(* Logix 5000 project; controller DispersionPlc vendor 1 type 14 code 108 rev 34.11; software revision 34.01; part 8 of 22 *)
(* tags used below, declared in another part *)
   Disp_Ons : BOOL[32];
   DispersionProductID_BarcodeScan : STRING;
   DispersionProductID_ScanIndex_Storage : DINT;
   DispersionProductIDEntryStorage : STRING;
   DispersionProductIDMatch : DINT;
   FE_4303_Deaband_Minus : REAL;
   FE_4303_Deaband_Plus : REAL;
   FE_4303_Feed_Error : REAL;
   FE_4303_Temp : REAL;
   Messaging_Timer2 : TIMER;
   MMI_SV4303_01_PB : BOOL;
   MMI_V4303_Acc_weight : REAL;
   MonDispenced_Snapshot : REAL;
   Monomer_FlowTimer : TIMER;
   Monomer_OneShots : BOOL[32];
   Monomer_Target_Wgt_Lb_Min : REAL;
   MonomerTimers : TIMER[12];
   ONS : BOOL[32];
   ons100 : BOOL;
   P4303_Rate : REAL;
   SV_4303_03_Man_Override : BOOL;
   T4301_T4302_Xfer_In_Enable : BOOL;
   W4303_RampTimer : TIMER;
   AFI : BOOL;
   BarcodeBypassAcitve : BOOL;
   BarcodeBypassAcitvePB : BOOL;
   BarcodeForEditString : STRING;
   BarcodeIndex : DINT;
   BarcodeIndex_Hold : DINT;
   BLANK64 : Stp64;
   BlankStrg : STRING;
   Cat_Tank_Destination : DINT;
   Control_Rm_tags : DINT;
   CR : STRING;
   CRADT : ALIAS FOR Local:5:O.Data.7;
   Dispersion_from_Main : DINT;
   Dispersion_from_Main2 : DINT;
   Dispersion_from_Main2_DintToStringConv : STRING;
   Dispersion_from_SIL2 : DINT;
   Dispersion_from_SIL2_Analog : REAL[24];
   Dispersion_to_Main : DINT;
   Dispersion_to_SIL2 : DINT;
   Dispersion_to_SIL2_Analog : REAL[24];
   DispersionAlarms : BOOL[256];
   DispersionProductID : STRING[21];
   DispersionProductID_ScanIndex : DINT;
   DispersionProductIDKeyEntry : STRING;
   DispersionProductIDKeyEntry1 : STRING;
   Drum_Transfer : BOOL;
   Drum_Transfer_Active : BOOL;
   Drum_Transfer_ONS : BOOL;
   Drum_Transfer_ONS_1 : BOOL;
   Enable_High_Alarm : BOOL;
   Enable_Shortstop_Automation : BOOL;
   Estop_Inx : ALIAS FOR Local:3:I.Data.3;
   FE_4303_Corrected : REAL;
   Found : DINT;
   From_Main : MESSAGE;
   From_Sil2 : MESSAGE;
   From_Sil2_Analog : MESSAGE;
   Hold_For_Flow_Switch : BOOL;
   Hold_For_Pump_Enable : BOOL;
   K4_High_Temp : BOOL;
   K4_Low_Temp : BOOL;
   LastScannedCode : STRING;
   LevelAlarmBeaconsRelay : BOOL;
   LS_26_High : BOOL;
   LS_28_H_Alarm : BOOL;
   MAINT_SV4303_03_PB : BOOL;
   MAINT_SV4303_04_PB : BOOL;
   MAINT_XV4303_05_PB : BOOL;
   Messaging_Timer : TIMER;
   MIXER_A_4303_RUN : ALIAS FOR Local:1:O.Data[0].4;
   MMI_A_4303_RUN_PB : BOOL;
   MMI_Mon_Nit_Purge_Time : REAL;
   MMI_Mon_Recirc_Pump_Speed : REAL;
   MMI_P_4303_Run_Pb : BOOL;
   MMI_SV4303_03_PB : BOOL;
   MMI_SV4303_04_PB : BOOL;
   MMI_V4303_Acc_Weight_Reset : BOOL;
   MMI_V4303_TransTime_SP : REAL;
   MMI_V4303_Weight_SP : REAL;
   MMI_W4303_Acc_Weight : REAL;
   MMI_XV4303_03_PB : BOOL;
   MMI_XV4303_04_PB : BOOL;
   MMI_XV4303_05_PB : BOOL;
   Momomer_Ons : DINT;
   Mon_Bogus_Bit : BOOL;
   Mon_Pump_Manual : BOOL;
   Mon_Recirc_Transfer_K400 : Seq64;
   Mon_Recirc_Transfer_T430X : Seq64;
   Mon_Tank_Destination : DINT;
   MON_VALV_ENBL : DINT;
   Monomer_Barcode : STRING;
   Monomer_Barcode_Scan_Index : DINT;
   Monomer_Barcode_Search : BOOL;
   Monomer_Fill_Pump_Running : BOOL;
   Monomer_Fill_Pump_Stopped : BOOL;
   Monomer_Flow_Start_Timer : TIMER;
   Monomer_Flow_Stop_Timer : TIMER;
   Monomer_MaxFeedRate : REAL;
   MONOMER_RESET : BOOL;
   Monomer_Scanner_Reset_Timer : TIMER;
   MonomerTimers_0_HMI : REAL;
   No_Vaild_Monomer_Barcode_Found : BOOL;
   One_Shots : DINT;
   OneShots : DINT;
   Pump_Enable_TMR : TIMER;
   SaveBarcode : BOOL;
   ScreenDisplayBarcode : STRING;
   Shortstop_Activate : BOOL;
   Shortstop_Timer_1 : REAL;
   Shortstop_Timer_2 : REAL;
   SIL2_to_Dispersion : DINT;
   SPARE_O515 : ALIAS FOR Local:5:O.Data.15;
   ST_K400_1 : REAL;
   ST_K400_SAFETY : BOOL;
   SV_4303_01 : ALIAS FOR Local:5:O.Data.8;
   SV_4303_02_ZSC : BOOL;
   SV_4303_02_ZSO : BOOL;
   SV_4303_03 : BOOL;
   SV_4303_03_Enable_PB : BOOL;
   SV_4303_04 : BOOL;
   SV_4303_04_Enable_PB : BOOL;
   T4301_Mixer : VFD;
   T4301_Process_Alarm_Setpoints : Alarm_SPT;
   Task_Permissive : DINT[2];
   TE_4301A : ALIAS FOR Local:8:I.Ch0Data;
   TE_4303_01 : REAL;
   TE_4303_High : REAL;
   To_CtrlRm1 : MESSAGE;
   To_CtrlRm2 : MESSAGE;
   To_CtrlRm3 : MESSAGE;
   To_Main : MESSAGE;
   To_Main2 : MESSAGE;
   To_SIL2 : MESSAGE;
   To_SIL2_Analog : MESSAGE;
   TOGGLE : BOOL;
   TruckLoadLevelAlarmHIHI : BOOL;
   TruckLoadLevelAlarmHIHIRedundant : BOOL;
   TruckLoadLevelAlarmResetPB : BOOL;
   V4304_Pump : VFD;
   Vaild_Monomer_Barcode : BOOL;
   Vaild_Monomer_Barcode_At_Index : DINT;
   Vaild_Monomer_BarcodeS : STRING[20];
   W4303_Pump : VFD;
   XI_K400_1 : BOOL;
   XV_4303_01 : ALIAS FOR Local:5:O.Data.3;
   XV_4303_01_PB : BOOL;
   XV_4303_02_ZSC : BOOL;
   XV_4303_02_ZSO : BOOL;
   XV_4303_03 : BOOL;
   XV_4303_04 : BOOL;
   XV_4303_05 : BOOL;
   XV_K400_03_SEQCLOSE : BOOL;
   XV_K400_03_SEQOPEN : BOOL;
   XV_K400_04_SEQCLOSE : BOOL;
   XV_K400_04_SEQOPEN : BOOL;
   ZSC_4303_03 : BOOL;
   ZSC_4303_04 : BOOL;
   ZSC_4303_05 : BOOL;
   ZSC_4303_1 : ALIAS FOR Local:2:I.Data.7;
   ZSC_K400_03 : BOOL;
   ZSC_K400_04 : BOOL;
   ZSO_4303_04 : BOOL;
   ZSO_4303_05 : BOOL;
   ZSO_K400_03 : BOOL;
   ZSO_K400_04 : BOOL;
(* MainProgram, continued *)

ROUTINE Messaging   (* ladder *)
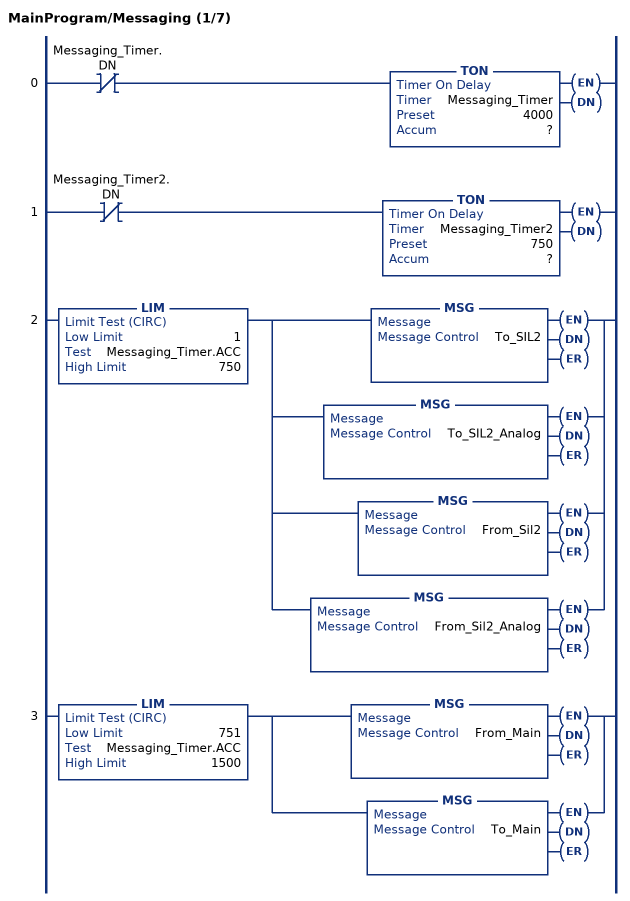
   0: XIO(Messaging_Timer.DN)TON(Messaging_Timer,?,?);
   1: XIO(Messaging_Timer2.DN)TON(Messaging_Timer2,?,?);
   2: LIM(1,Messaging_Timer.ACC,750)[MSG(To_SIL2) ,MSG(To_SIL2_Analog) ,MSG(From_Sil2) ,MSG(From_Sil2_Analog) ];
   3: LIM(751,Messaging_Timer.ACC,1500)[MSG(From_Main) ,MSG(To_Main) ];
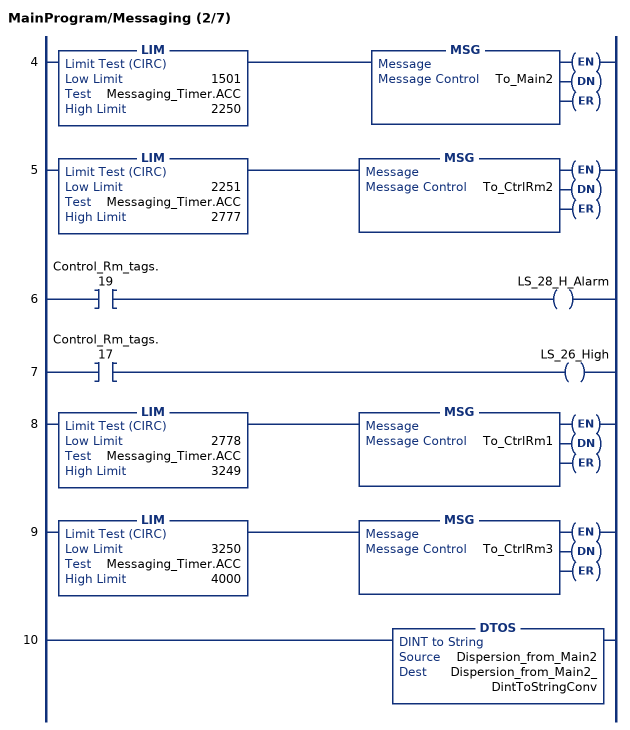
   4: LIM(1501,Messaging_Timer.ACC,2250)MSG(To_Main2);
   5: LIM(2251,Messaging_Timer.ACC,2777)MSG(To_CtrlRm2);
   6: XIC(Control_Rm_tags.19)OTE(LS_28_H_Alarm);
   7: XIC(Control_Rm_tags.17)OTE(LS_26_High);
   8: LIM(2778,Messaging_Timer.ACC,3249)MSG(To_CtrlRm1);
   9: LIM(3250,Messaging_Timer.ACC,4000)MSG(To_CtrlRm3);
   10: DTOS(Dispersion_from_Main2,Dispersion_from_Main2_DintToStringConv);
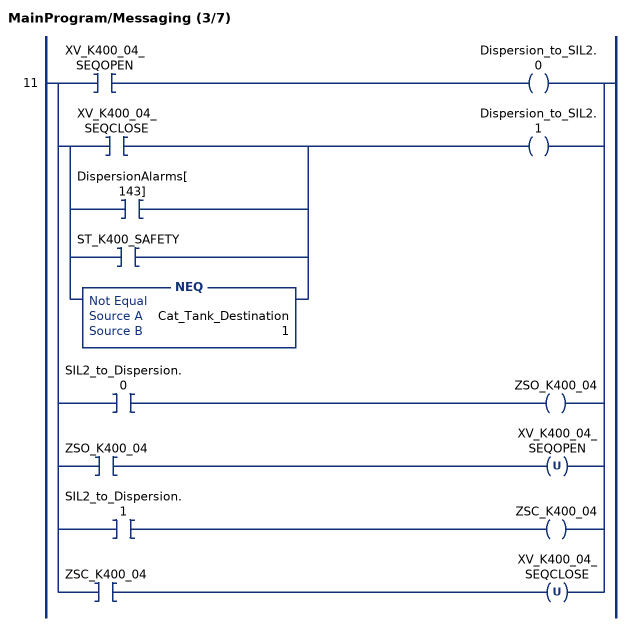
   11: [XIC(XV_K400_04_SEQOPEN) OTE(Dispersion_to_SIL2.0) ,[XIC(XV_K400_04_SEQCLOSE) ,XIC(DispersionAlarms[143]) ,XIC(ST_K400_SAFETY) ,NEQ(Cat_Tank_Destination,1) ] OTE(Dispersion_to_SIL2.1) ,XIC(SIL2_to_Dispersion.0) OTE(ZSO_K400_04) ,XIC(ZSO_K400_04) OTU(XV_K400_04_SEQOPEN) ,XIC(SIL2_to_Dispersion.1) OTE(ZSC_K400_04) ,XIC(ZSC_K400_04) OTU(XV_K400_04_SEQCLOSE) ];
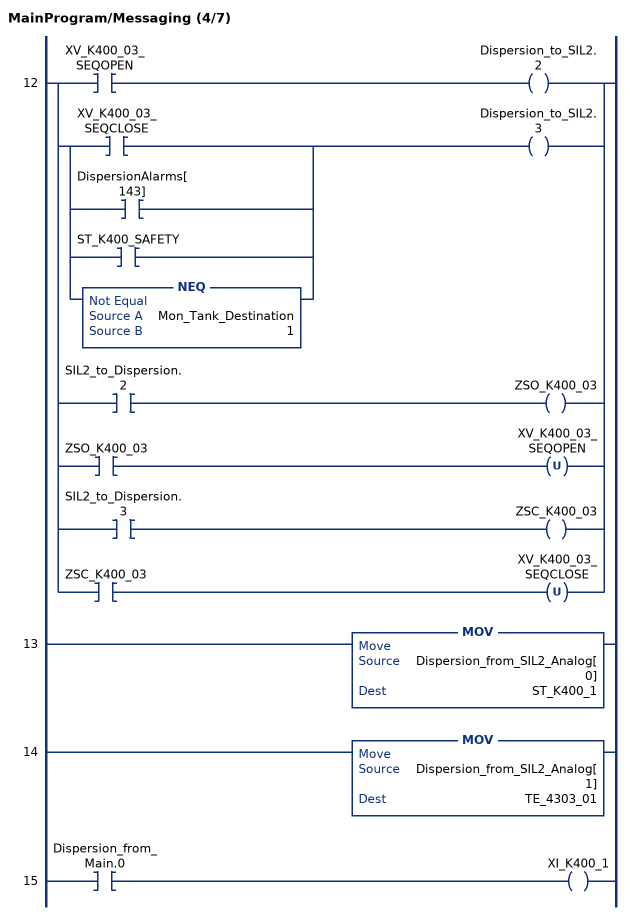
   12: [XIC(XV_K400_03_SEQOPEN) OTE(Dispersion_to_SIL2.2) ,[XIC(XV_K400_03_SEQCLOSE) ,XIC(DispersionAlarms[143]) ,XIC(ST_K400_SAFETY) ,NEQ(Mon_Tank_Destination,1) ] OTE(Dispersion_to_SIL2.3) ,XIC(SIL2_to_Dispersion.2) OTE(ZSO_K400_03) ,XIC(ZSO_K400_03) OTU(XV_K400_03_SEQOPEN) ,XIC(SIL2_to_Dispersion.3) OTE(ZSC_K400_03) ,XIC(ZSC_K400_03) OTU(XV_K400_03_SEQCLOSE) ];
   13: MOV(Dispersion_from_SIL2_Analog[0],ST_K400_1);
   14: MOV(Dispersion_from_SIL2_Analog[1],TE_4303_01);
   15: XIC(Dispersion_from_Main.0)OTE(XI_K400_1);
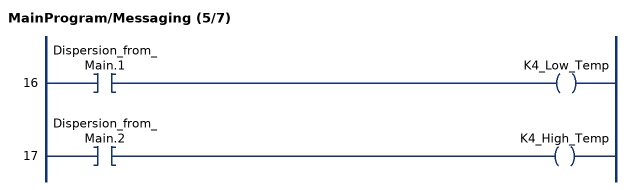
   16: XIC(Dispersion_from_Main.1)OTE(K4_Low_Temp);
   17: XIC(Dispersion_from_Main.2)OTE(K4_High_Temp);
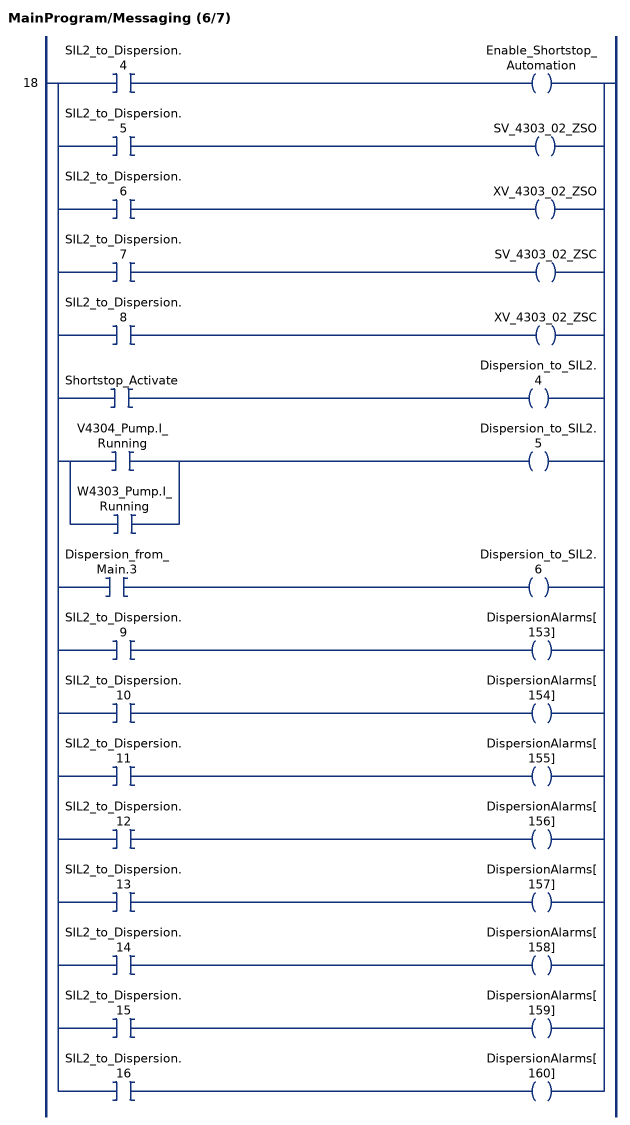
   18: [XIC(SIL2_to_Dispersion.4) OTE(Enable_Shortstop_Automation) ,XIC(SIL2_to_Dispersion.5) OTE(SV_4303_02_ZSO) ,XIC(SIL2_to_Dispersion.6) OTE(XV_4303_02_ZSO) ,XIC(SIL2_to_Dispersion.7) OTE(SV_4303_02_ZSC) ,XIC(SIL2_to_Dispersion.8) OTE(XV_4303_02_ZSC) ,XIC(Shortstop_Activate) OTE(Dispersion_to_SIL2.4) ,[XIC(V4304_Pump.I_Running) ,XIC(W4303_Pump.I_Running) ] OTE(Dispersion_to_SIL2.5) ,XIC(Dispersion_from_Main.3) OTE(Dispersion_to_SIL2.6) ,XIC(SIL2_to_Dispersion.9) OTE(DispersionAlarms[153]) ,XIC(SIL2_to_Dispersion.10) OTE(DispersionAlarms[154]) ,XIC(SIL2_to_Dispersion.11) OTE(DispersionAlarms[155]) ,XIC(SIL2_to_Dispersion.12) OTE(DispersionAlarms[156]) ,XIC(SIL2_to_Dispersion.13) OTE(DispersionAlarms[157]) ,XIC(SIL2_to_Dispersion.14) OTE(DispersionAlarms[158]) ,XIC(SIL2_to_Dispersion.15) OTE(DispersionAlarms[159]) ,XIC(SIL2_to_Dispersion.16) OTE(DispersionAlarms[160]) ];
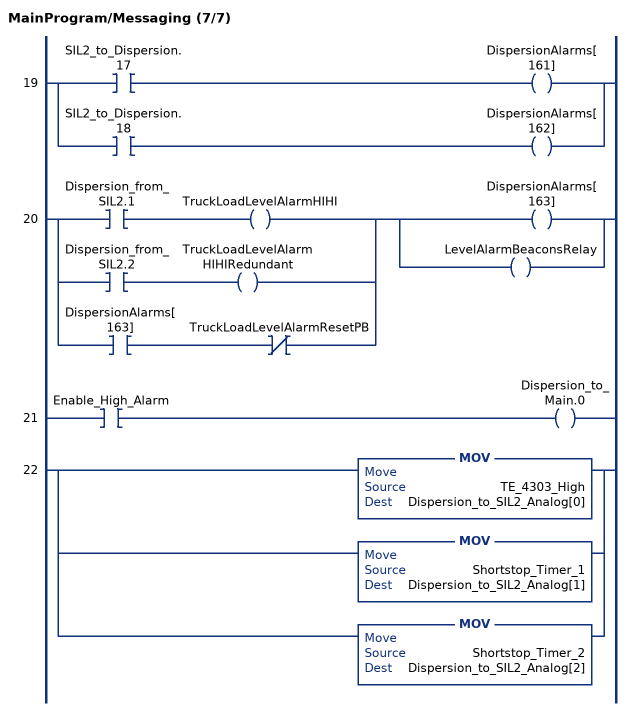
   19: [XIC(SIL2_to_Dispersion.17) OTE(DispersionAlarms[161]) ,XIC(SIL2_to_Dispersion.18) OTE(DispersionAlarms[162]) ];
   20: [[XIC(Dispersion_from_SIL2.1) OTE(TruckLoadLevelAlarmHIHI) ,XIC(Dispersion_from_SIL2.2) OTE(TruckLoadLevelAlarmHIHIRedundant) ] ,XIC(DispersionAlarms[163]) XIO(TruckLoadLevelAlarmResetPB) ][OTE(DispersionAlarms[163]) ,OTE(LevelAlarmBeaconsRelay) ];
   21: XIC(Enable_High_Alarm)OTE(Dispersion_to_Main.0);
   22: [MOV(TE_4303_High,Dispersion_to_SIL2_Analog[0]) ,MOV(Shortstop_Timer_1,Dispersion_to_SIL2_Analog[1]) ,MOV(Shortstop_Timer_2,Dispersion_to_SIL2_Analog[2]) ];
END_ROUTINE

ROUTINE Monomer   (* ladder *)
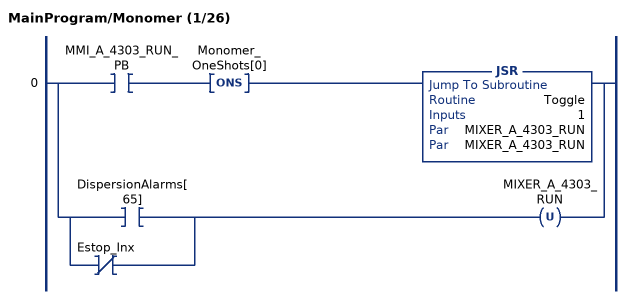
   0: [XIC(MMI_A_4303_RUN_PB) ONS(Monomer_OneShots[0]) JSR(Toggle,1,MIXER_A_4303_RUN,MIXER_A_4303_RUN) ,[XIC(DispersionAlarms[65]) ,XIO(Estop_Inx) ] OTU(MIXER_A_4303_RUN) ];
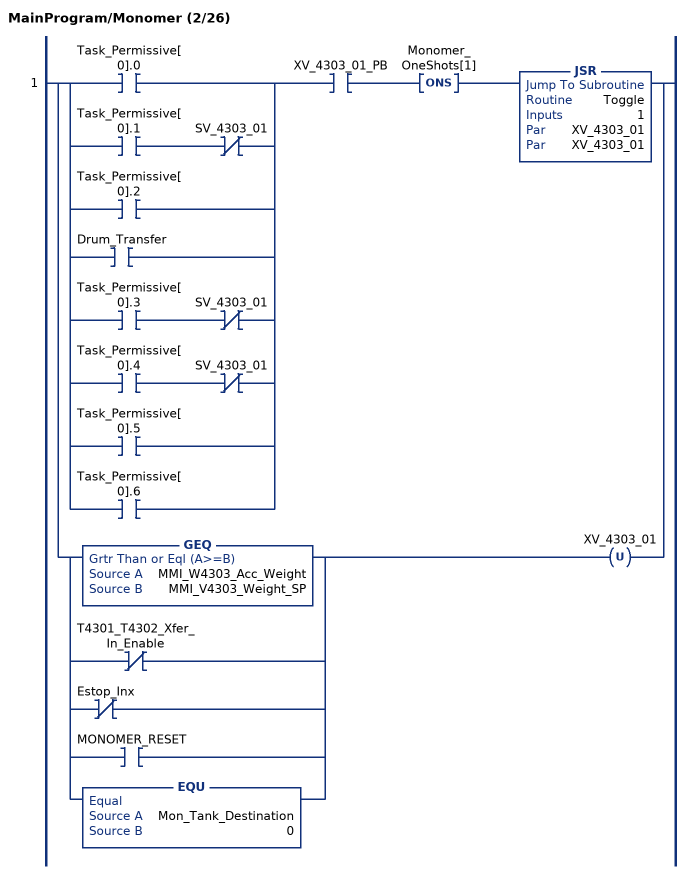
   1: [[XIC(Task_Permissive[0].0) ,XIC(Task_Permissive[0].1) XIO(SV_4303_01) ,XIC(Task_Permissive[0].2) ,XIC(Drum_Transfer) ,XIC(Task_Permissive[0].3) XIO(SV_4303_01) ,XIC(Task_Permissive[0].4) XIO(SV_4303_01) ,XIC(Task_Permissive[0].5) ,XIC(Task_Permissive[0].6) ] XIC(XV_4303_01_PB) ONS(Monomer_OneShots[1]) JSR(Toggle,1,XV_4303_01,XV_4303_01) ,[GEQ(MMI_W4303_Acc_Weight,MMI_V4303_Weight_SP) ,XIO(T4301_T4302_Xfer_In_Enable) ,XIO(Estop_Inx) ,XIC(MONOMER_RESET) ,EQU(Mon_Tank_Destination,0) ] OTU(XV_4303_01) ];
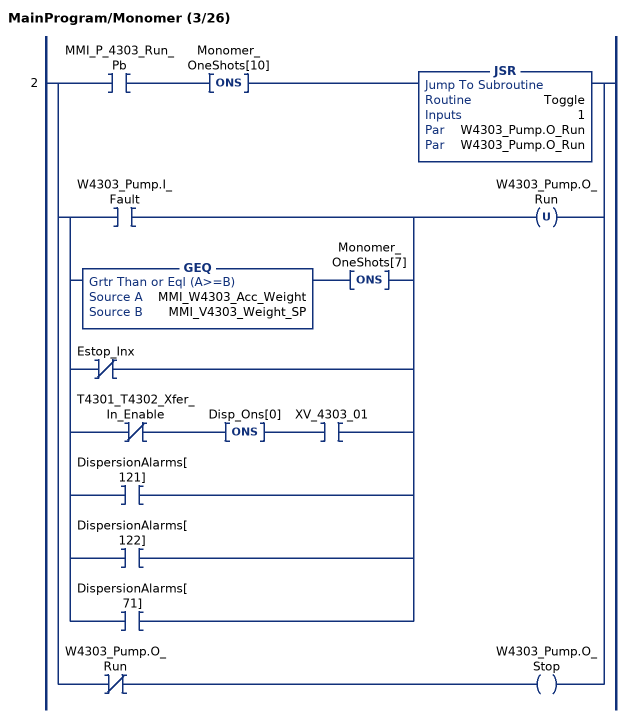
   2: [XIC(MMI_P_4303_Run_Pb) ONS(Monomer_OneShots[10]) JSR(Toggle,1,W4303_Pump.O_Run,W4303_Pump.O_Run) ,[XIC(W4303_Pump.I_Fault) ,GEQ(MMI_W4303_Acc_Weight,MMI_V4303_Weight_SP) ONS(Monomer_OneShots[7]) ,XIO(Estop_Inx) ,XIO(T4301_T4302_Xfer_In_Enable) ONS(Disp_Ons[0]) XIC(XV_4303_01) ,XIC(DispersionAlarms[121]) ,XIC(DispersionAlarms[122]) ,XIC(DispersionAlarms[71]) ] OTU(W4303_Pump.O_Run) ,XIO(W4303_Pump.O_Run) OTE(W4303_Pump.O_Stop) ];
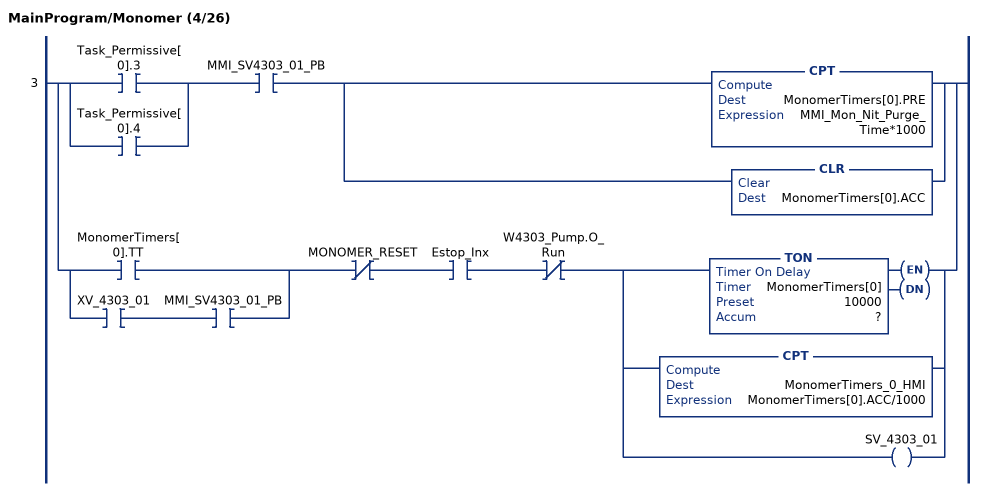
   3: [[XIC(Task_Permissive[0].3) ,XIC(Task_Permissive[0].4) ] XIC(MMI_SV4303_01_PB) [CPT(MonomerTimers[0].PRE,MMI_Mon_Nit_Purge_Time*1000) ,CLR(MonomerTimers[0].ACC) ] ,[XIC(MonomerTimers[0].TT) ,XIC(XV_4303_01) XIC(MMI_SV4303_01_PB) ] XIO(MONOMER_RESET) XIC(Estop_Inx) XIO(W4303_Pump.O_Run) [[TON(MonomerTimers[0],?,?) ,CPT(MonomerTimers_0_HMI,MonomerTimers[0].ACC/1000) ] ,OTE(SV_4303_01) ] ];
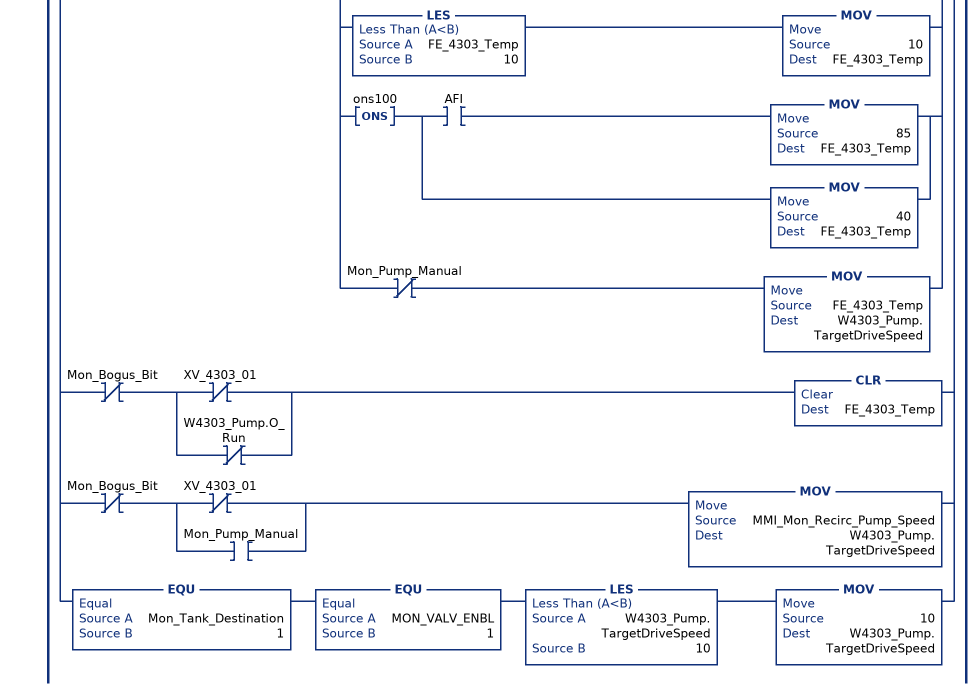
   4: [XIC(MMI_V4303_Acc_Weight_Reset) [CLR(MMI_W4303_Acc_Weight) ,OTU(MMI_V4303_Acc_Weight_Reset) ] ,LEQ(MMI_V4303_TransTime_SP,1) MOV(1,MMI_V4303_TransTime_SP) ,DIV(MMI_V4303_Weight_SP,MMI_V4303_TransTime_SP,Monomer_Target_Wgt_Lb_Min) ,GRT(Monomer_Target_Wgt_Lb_Min,Monomer_MaxFeedRate) MOV(Monomer_MaxFeedRate,Monomer_Target_Wgt_Lb_Min) ,SUB(FE_4303_Corrected,Monomer_Target_Wgt_Lb_Min,FE_4303_Feed_Error) ,[XIC(XV_4303_01) ,XIC(Mon_Bogus_Bit) ,XIC(Mon_Pump_Manual) ] XIC(W4303_Pump.O_Run) [XIO(W4303_RampTimer.DN) TON(W4303_RampTimer,?,?) ,XIC(W4303_RampTimer.DN) [CPT(MMI_W4303_Acc_Weight,MMI_W4303_Acc_Weight+(FE_4303_Corrected/(60/(W4303_RampTimer.PRE*0.001)))) ,LES(FE_4303_Feed_Error,FE_4303_Deaband_Minus) ADD(FE_4303_Temp,P4303_Rate,FE_4303_Temp) ,GRT(FE_4303_Feed_Error,FE_4303_Deaband_Plus) SUB(FE_4303_Temp,P4303_Rate,FE_4303_Temp) ] ,GRT(FE_4303_Temp,100) MOV(100,FE_4303_Temp) ,LES(FE_4303_Temp,10) MOV(10,FE_4303_Temp) ,ONS(ons100) [XIC(AFI) MOV(85,FE_4303_Temp) ,MOV(40,FE_4303_Temp) ] ,XIO(Mon_Pump_Manual) MOV(FE_4303_Temp,W4303_Pump.TargetDriveSpeed) ] ,XIO(Mon_Bogus_Bit) [XIO(XV_4303_01) ,XIO(W4303_Pump.O_Run) ] CLR(FE_4303_Temp) ,XIO(Mon_Bogus_Bit) [XIO(XV_4303_01) ,XIC(Mon_Pump_Manual) ] MOV(MMI_Mon_Recirc_Pump_Speed,W4303_Pump.TargetDriveSpeed) ,EQU(Mon_Tank_Destination,1) EQU(MON_VALV_ENBL,1) LES(W4303_Pump.TargetDriveSpeed,10) MOV(10,W4303_Pump.TargetDriveSpeed) ];
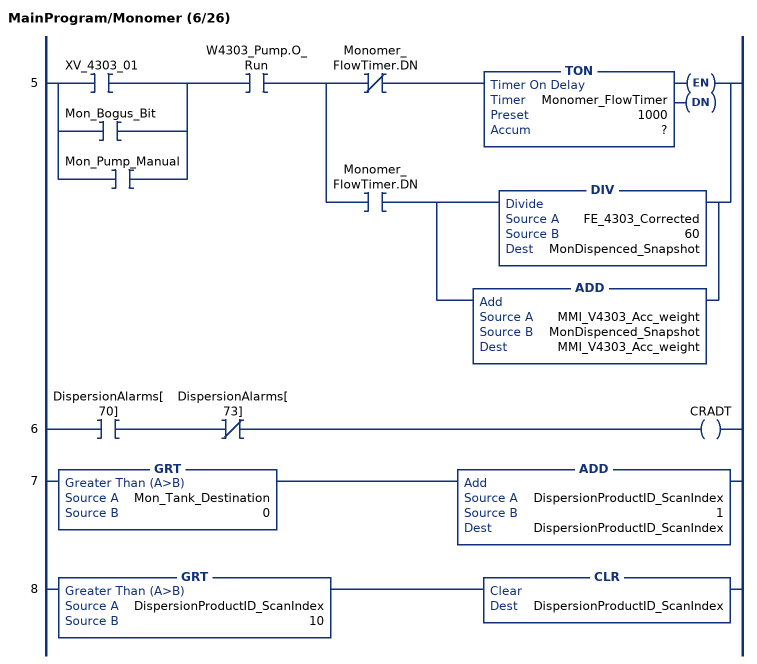
   5: [XIC(XV_4303_01) ,XIC(Mon_Bogus_Bit) ,XIC(Mon_Pump_Manual) ]XIC(W4303_Pump.O_Run)[XIO(Monomer_FlowTimer.DN) TON(Monomer_FlowTimer,?,?) ,XIC(Monomer_FlowTimer.DN) [DIV(FE_4303_Corrected,60,MonDispenced_Snapshot) ,ADD(MMI_V4303_Acc_weight,MonDispenced_Snapshot,MMI_V4303_Acc_weight) ] ];
   6: XIC(DispersionAlarms[70])XIO(DispersionAlarms[73])OTE(CRADT);
   7: GRT(Mon_Tank_Destination,0)ADD(DispersionProductID_ScanIndex,1,DispersionProductID_ScanIndex);
   8: GRT(DispersionProductID_ScanIndex,10)CLR(DispersionProductID_ScanIndex);
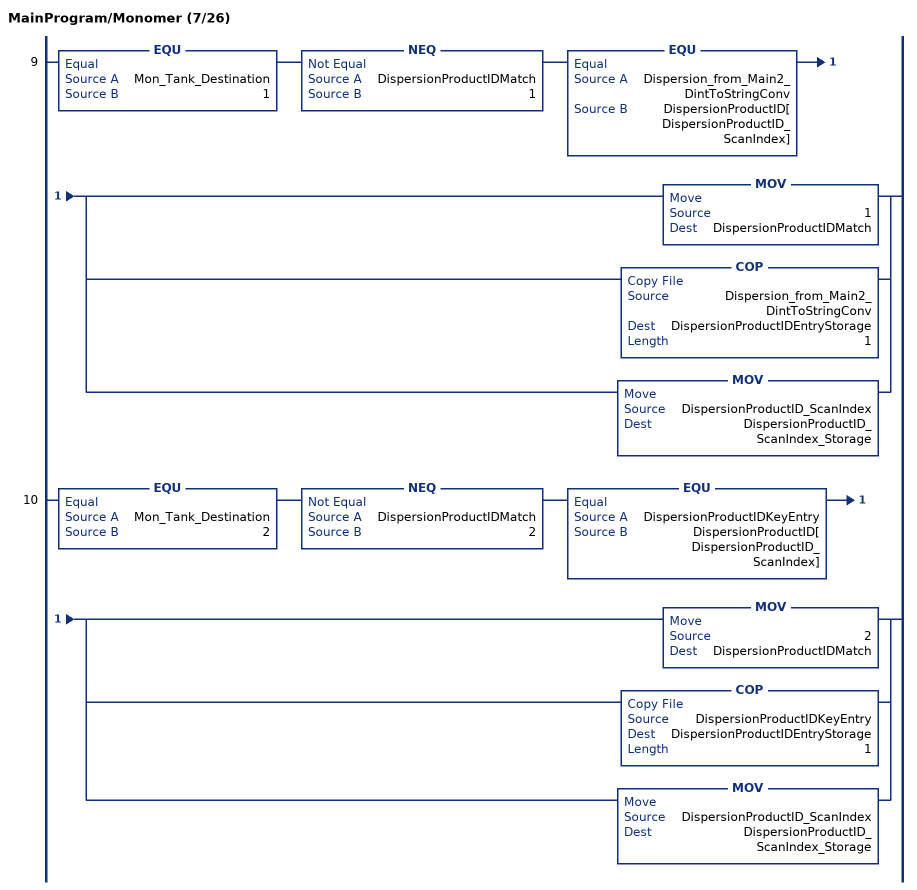
   9: EQU(Mon_Tank_Destination,1)NEQ(DispersionProductIDMatch,1)EQU(Dispersion_from_Main2_DintToStringConv,DispersionProductID[DispersionProductID_ScanIndex])[MOV(1,DispersionProductIDMatch) ,COP(Dispersion_from_Main2_DintToStringConv,DispersionProductIDEntryStorage,1) ,MOV(DispersionProductID_ScanIndex,DispersionProductID_ScanIndex_Storage) ];
   10: EQU(Mon_Tank_Destination,2)NEQ(DispersionProductIDMatch,2)EQU(DispersionProductIDKeyEntry,DispersionProductID[DispersionProductID_ScanIndex])[MOV(2,DispersionProductIDMatch) ,COP(DispersionProductIDKeyEntry,DispersionProductIDEntryStorage,1) ,MOV(DispersionProductID_ScanIndex,DispersionProductID_ScanIndex_Storage) ];
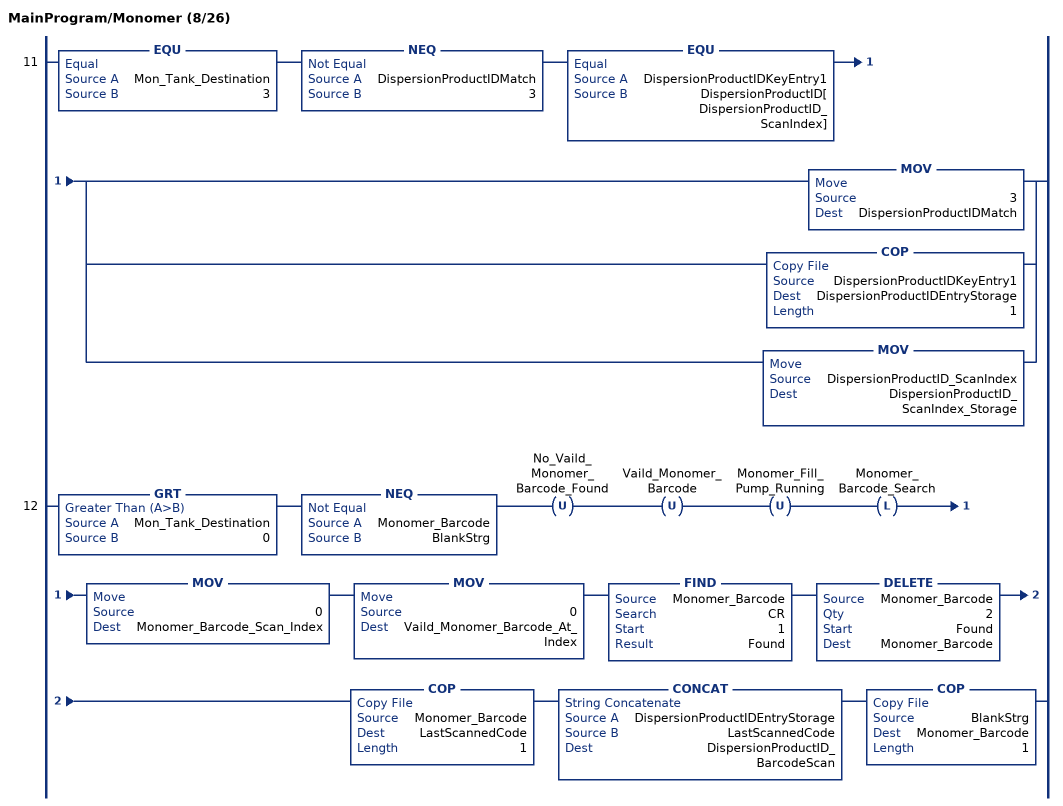
   11: EQU(Mon_Tank_Destination,3)NEQ(DispersionProductIDMatch,3)EQU(DispersionProductIDKeyEntry1,DispersionProductID[DispersionProductID_ScanIndex])[MOV(3,DispersionProductIDMatch) ,COP(DispersionProductIDKeyEntry1,DispersionProductIDEntryStorage,1) ,MOV(DispersionProductID_ScanIndex,DispersionProductID_ScanIndex_Storage) ];
   12: GRT(Mon_Tank_Destination,0)NEQ(Monomer_Barcode,BlankStrg)OTU(No_Vaild_Monomer_Barcode_Found)OTU(Vaild_Monomer_Barcode)OTU(Monomer_Fill_Pump_Running)OTL(Monomer_Barcode_Search)MOV(0,Monomer_Barcode_Scan_Index)MOV(0,Vaild_Monomer_Barcode_At_Index)FIND(Monomer_Barcode,CR,1,Found)DELETE(Monomer_Barcode,2,Found,Monomer_Barcode)COP(Monomer_Barcode,LastScannedCode,1)CONCAT(DispersionProductIDEntryStorage,LastScannedCode,DispersionProductID_BarcodeScan)COP(BlankStrg,Monomer_Barcode,1);
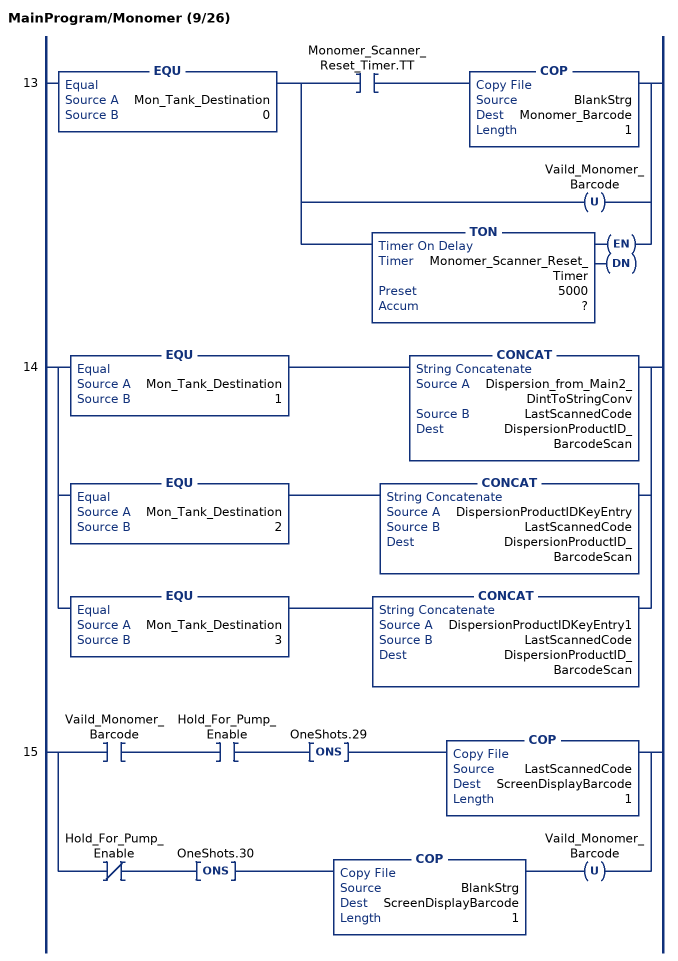
   13: EQU(Mon_Tank_Destination,0)[XIC(Monomer_Scanner_Reset_Timer.TT) COP(BlankStrg,Monomer_Barcode,1) ,OTU(Vaild_Monomer_Barcode) ,TON(Monomer_Scanner_Reset_Timer,?,?) ];
   14: [EQU(Mon_Tank_Destination,1) CONCAT(Dispersion_from_Main2_DintToStringConv,LastScannedCode,DispersionProductID_BarcodeScan) ,EQU(Mon_Tank_Destination,2) CONCAT(DispersionProductIDKeyEntry,LastScannedCode,DispersionProductID_BarcodeScan) ,EQU(Mon_Tank_Destination,3) CONCAT(DispersionProductIDKeyEntry1,LastScannedCode,DispersionProductID_BarcodeScan) ];
   15: [XIC(Vaild_Monomer_Barcode) XIC(Hold_For_Pump_Enable) ONS(OneShots.29) COP(LastScannedCode,ScreenDisplayBarcode,1) ,XIO(Hold_For_Pump_Enable) ONS(OneShots.30) COP(BlankStrg,ScreenDisplayBarcode,1) OTU(Vaild_Monomer_Barcode) ];
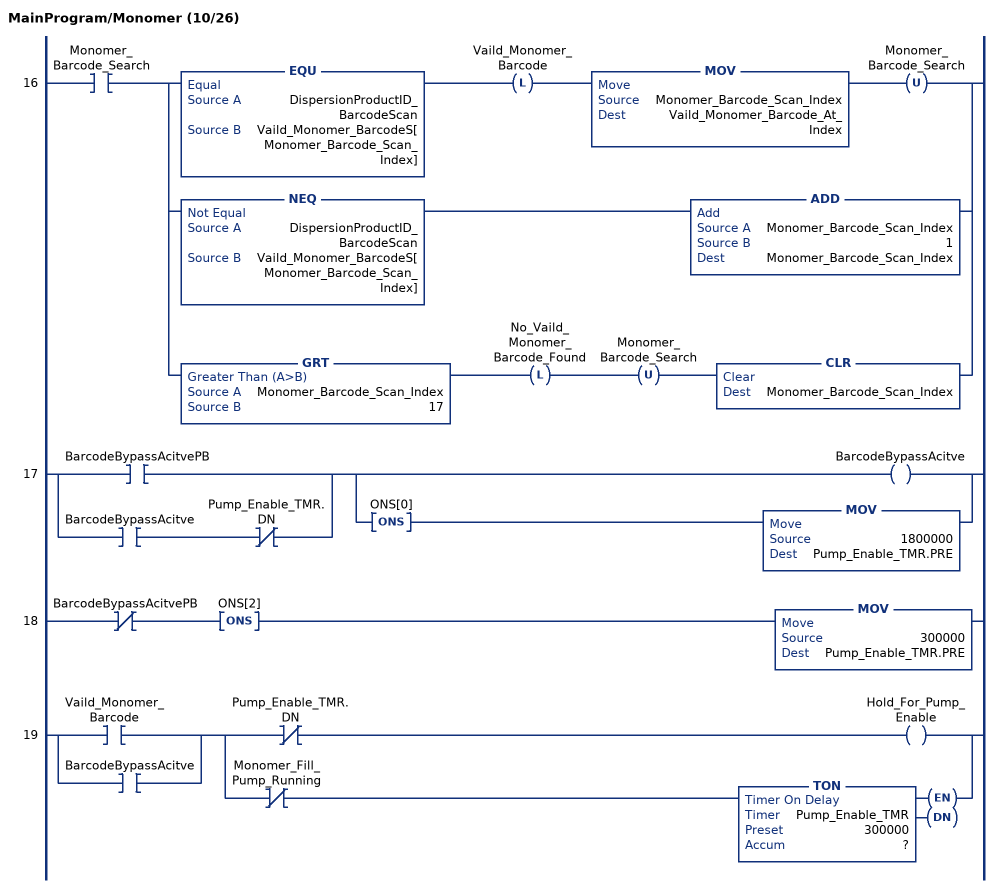
   16: XIC(Monomer_Barcode_Search)[EQU(DispersionProductID_BarcodeScan,Vaild_Monomer_BarcodeS[Monomer_Barcode_Scan_Index]) OTL(Vaild_Monomer_Barcode) MOV(Monomer_Barcode_Scan_Index,Vaild_Monomer_Barcode_At_Index) OTU(Monomer_Barcode_Search) ,NEQ(DispersionProductID_BarcodeScan,Vaild_Monomer_BarcodeS[Monomer_Barcode_Scan_Index]) ADD(Monomer_Barcode_Scan_Index,1,Monomer_Barcode_Scan_Index) ,GRT(Monomer_Barcode_Scan_Index,17) OTL(No_Vaild_Monomer_Barcode_Found) OTU(Monomer_Barcode_Search) CLR(Monomer_Barcode_Scan_Index) ];
   17: [XIC(BarcodeBypassAcitvePB) ,XIC(BarcodeBypassAcitve) XIO(Pump_Enable_TMR.DN) ][OTE(BarcodeBypassAcitve) ,ONS(ONS[0]) MOV(1800000,Pump_Enable_TMR.PRE) ];
   18: XIO(BarcodeBypassAcitvePB)ONS(ONS[2])MOV(300000,Pump_Enable_TMR.PRE);
   19: [XIC(Vaild_Monomer_Barcode) ,XIC(BarcodeBypassAcitve) ][XIO(Pump_Enable_TMR.DN) OTE(Hold_For_Pump_Enable) ,XIO(Monomer_Fill_Pump_Running) TON(Pump_Enable_TMR,?,?) ];
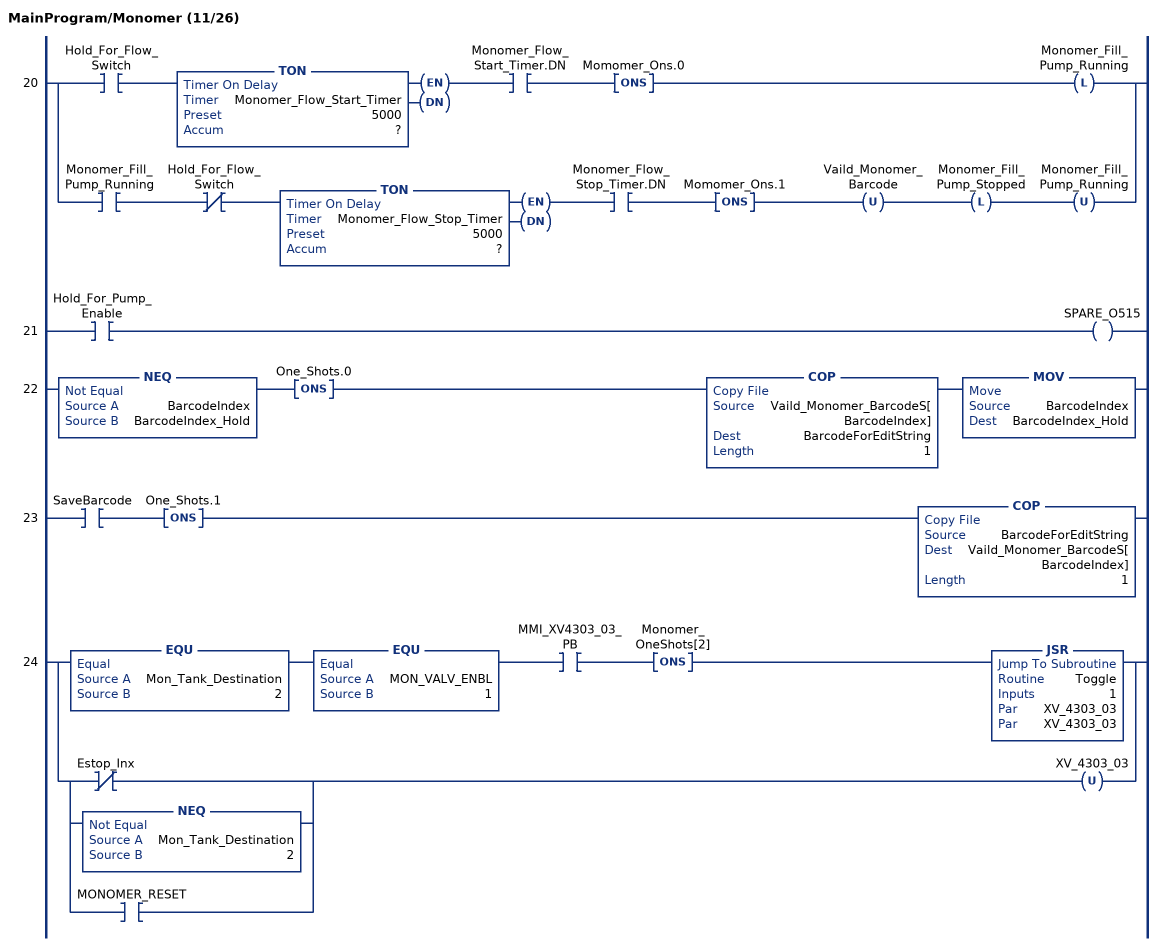
   20: [XIC(Hold_For_Flow_Switch) TON(Monomer_Flow_Start_Timer,?,?) XIC(Monomer_Flow_Start_Timer.DN) ONS(Momomer_Ons.0) OTL(Monomer_Fill_Pump_Running) ,XIC(Monomer_Fill_Pump_Running) XIO(Hold_For_Flow_Switch) TON(Monomer_Flow_Stop_Timer,?,?) XIC(Monomer_Flow_Stop_Timer.DN) ONS(Momomer_Ons.1) OTU(Vaild_Monomer_Barcode) OTL(Monomer_Fill_Pump_Stopped) OTU(Monomer_Fill_Pump_Running) ];
   21: XIC(Hold_For_Pump_Enable)OTE(SPARE_O515);
   22: NEQ(BarcodeIndex,BarcodeIndex_Hold)ONS(One_Shots.0)COP(Vaild_Monomer_BarcodeS[BarcodeIndex],BarcodeForEditString,1)MOV(BarcodeIndex,BarcodeIndex_Hold);
   23: XIC(SaveBarcode)ONS(One_Shots.1)COP(BarcodeForEditString,Vaild_Monomer_BarcodeS[BarcodeIndex],1);
   24: [EQU(Mon_Tank_Destination,2) EQU(MON_VALV_ENBL,1) XIC(MMI_XV4303_03_PB) ONS(Monomer_OneShots[2]) JSR(Toggle,1,XV_4303_03,XV_4303_03) ,[XIO(Estop_Inx) ,NEQ(Mon_Tank_Destination,2) ,XIC(MONOMER_RESET) ] OTU(XV_4303_03) ];
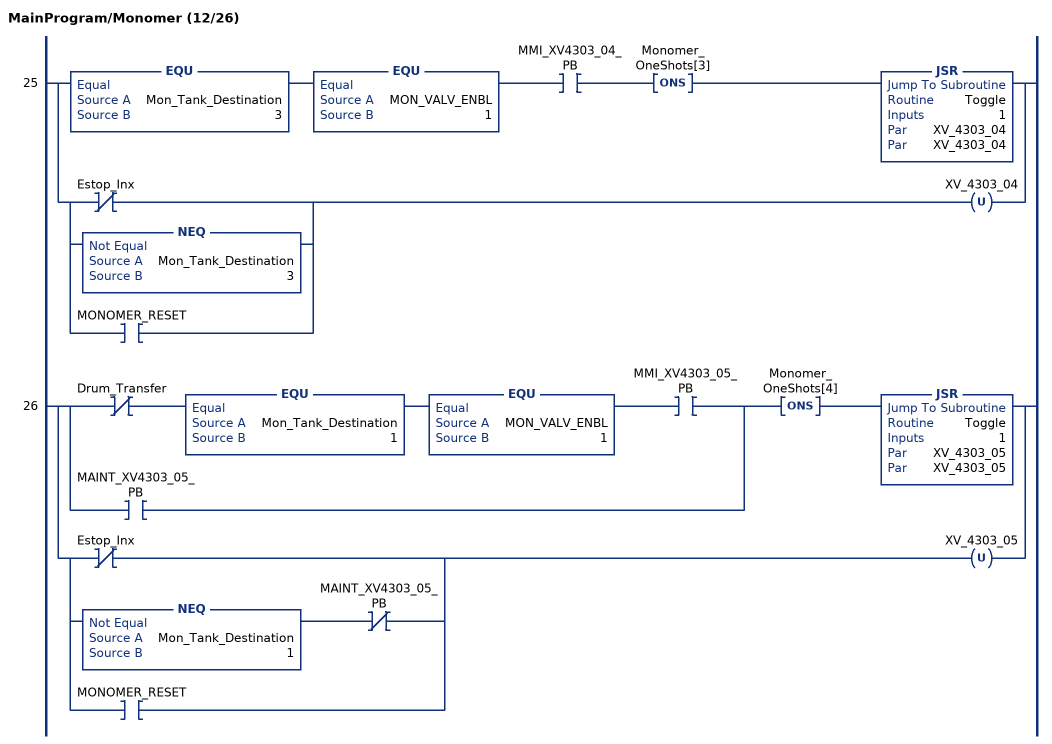
   25: [EQU(Mon_Tank_Destination,3) EQU(MON_VALV_ENBL,1) XIC(MMI_XV4303_04_PB) ONS(Monomer_OneShots[3]) JSR(Toggle,1,XV_4303_04,XV_4303_04) ,[XIO(Estop_Inx) ,NEQ(Mon_Tank_Destination,3) ,XIC(MONOMER_RESET) ] OTU(XV_4303_04) ];
   26: [[XIO(Drum_Transfer) EQU(Mon_Tank_Destination,1) EQU(MON_VALV_ENBL,1) XIC(MMI_XV4303_05_PB) ,XIC(MAINT_XV4303_05_PB) ] ONS(Monomer_OneShots[4]) JSR(Toggle,1,XV_4303_05,XV_4303_05) ,[XIO(Estop_Inx) ,NEQ(Mon_Tank_Destination,1) XIO(MAINT_XV4303_05_PB) ,XIC(MONOMER_RESET) ] OTU(XV_4303_05) ];
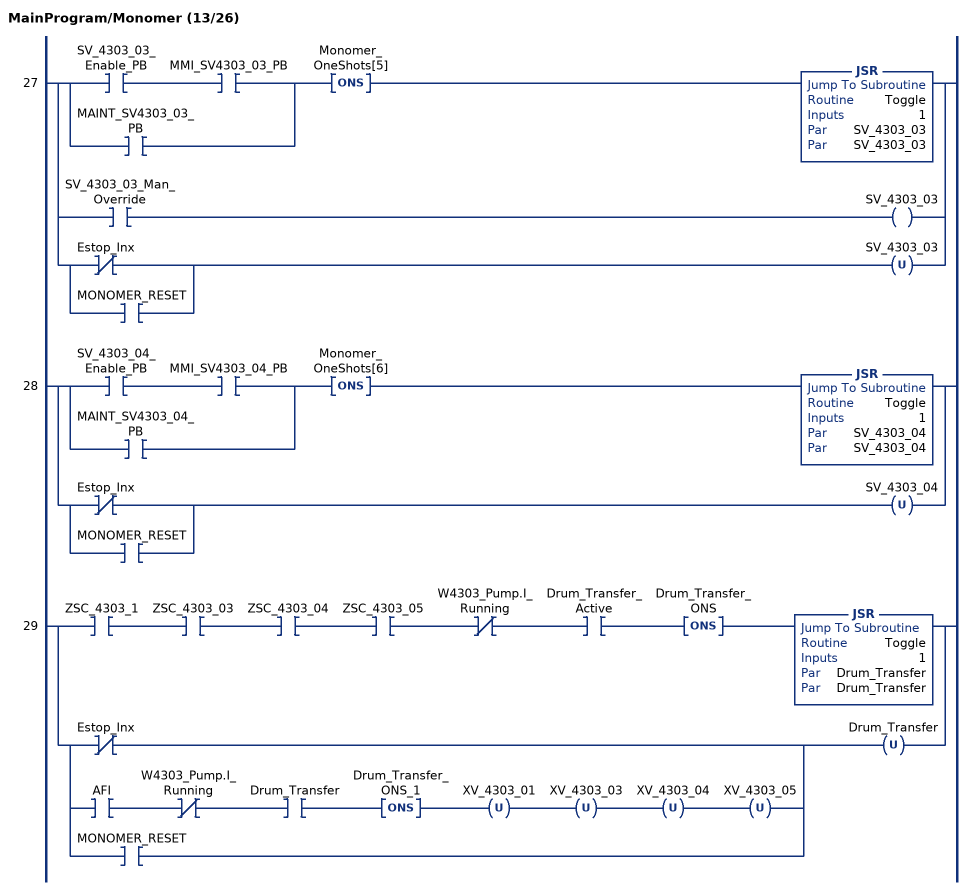
   27: [[[XIC(SV_4303_03_Enable_PB) XIC(MMI_SV4303_03_PB) ,XIC(MAINT_SV4303_03_PB) ] ONS(Monomer_OneShots[5]) JSR(Toggle,1,SV_4303_03,SV_4303_03) ,XIC(SV_4303_03_Man_Override) OTE(SV_4303_03) ] ,[XIO(Estop_Inx) ,XIC(MONOMER_RESET) ] OTU(SV_4303_03) ];
   28: [[XIC(SV_4303_04_Enable_PB) XIC(MMI_SV4303_04_PB) ,XIC(MAINT_SV4303_04_PB) ] ONS(Monomer_OneShots[6]) JSR(Toggle,1,SV_4303_04,SV_4303_04) ,[XIO(Estop_Inx) ,XIC(MONOMER_RESET) ] OTU(SV_4303_04) ];
   29: [XIC(ZSC_4303_1) XIC(ZSC_4303_03) XIC(ZSC_4303_04) XIC(ZSC_4303_05) XIO(W4303_Pump.I_Running) XIC(Drum_Transfer_Active) ONS(Drum_Transfer_ONS) JSR(Toggle,1,Drum_Transfer,Drum_Transfer) ,[XIO(Estop_Inx) ,XIC(AFI) XIO(W4303_Pump.I_Running) XIC(Drum_Transfer) ONS(Drum_Transfer_ONS_1) OTU(XV_4303_01) OTU(XV_4303_03) OTU(XV_4303_04) OTU(XV_4303_05) ,XIC(MONOMER_RESET) ] OTU(Drum_Transfer) ];
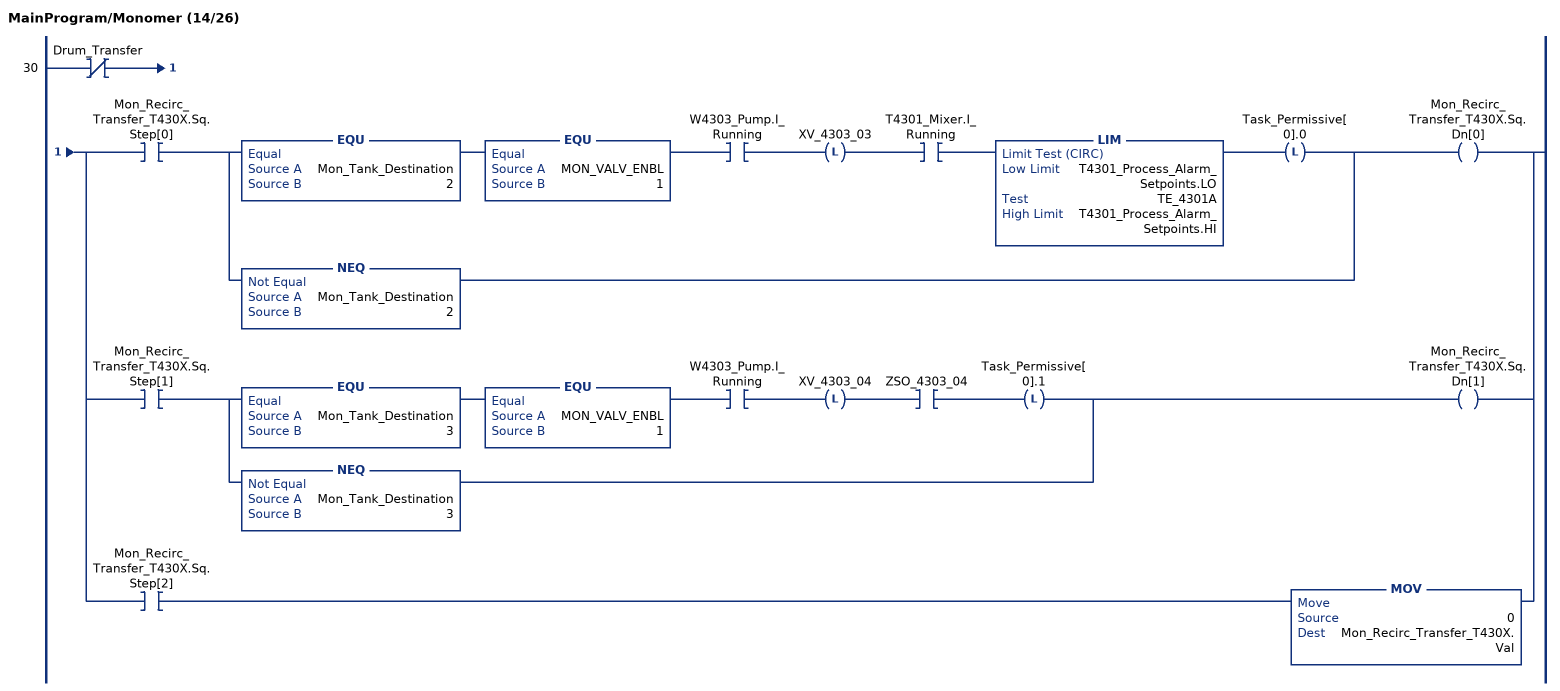
   30: XIO(Drum_Transfer)[XIC(Mon_Recirc_Transfer_T430X.Sq.Step[0]) [EQU(Mon_Tank_Destination,2) EQU(MON_VALV_ENBL,1) XIC(W4303_Pump.I_Running) OTL(XV_4303_03) XIC(T4301_Mixer.I_Running) LIM(T4301_Process_Alarm_Setpoints.LO,TE_4301A,T4301_Process_Alarm_Setpoints.HI) OTL(Task_Permissive[0].0) ,NEQ(Mon_Tank_Destination,2) ] OTE(Mon_Recirc_Transfer_T430X.Sq.Dn[0]) ,XIC(Mon_Recirc_Transfer_T430X.Sq.Step[1]) [EQU(Mon_Tank_Destination,3) EQU(MON_VALV_ENBL,1) XIC(W4303_Pump.I_Running) OTL(XV_4303_04) XIC(ZSO_4303_04) OTL(Task_Permissive[0].1) ,NEQ(Mon_Tank_Destination,3) ] OTE(Mon_Recirc_Transfer_T430X.Sq.Dn[1]) ,XIC(Mon_Recirc_Transfer_T430X.Sq.Step[2]) MOV(0,Mon_Recirc_Transfer_T430X.Val) ];
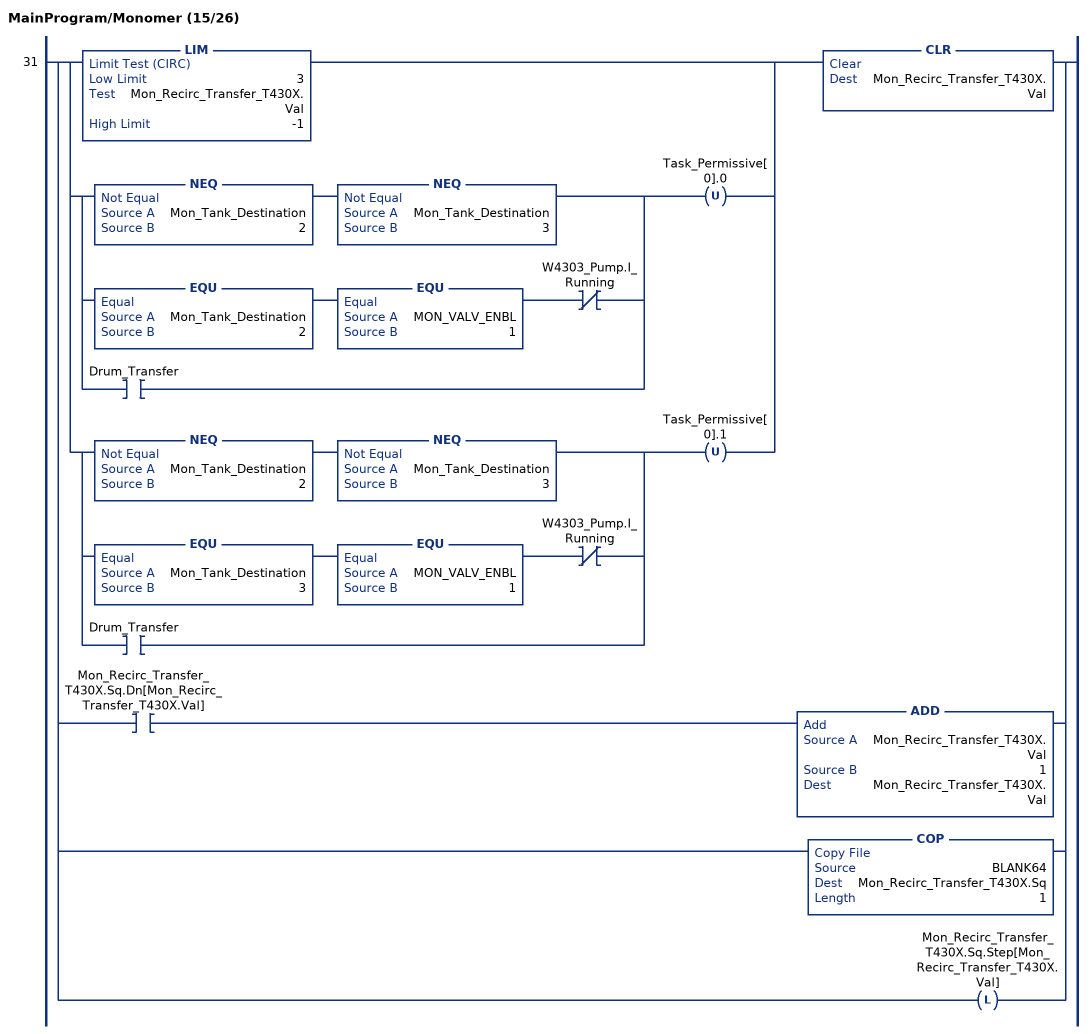
   31: [[LIM(3,Mon_Recirc_Transfer_T430X.Val,-1) ,[NEQ(Mon_Tank_Destination,2) NEQ(Mon_Tank_Destination,3) ,EQU(Mon_Tank_Destination,2) EQU(MON_VALV_ENBL,1) XIO(W4303_Pump.I_Running) ,XIC(Drum_Transfer) ] OTU(Task_Permissive[0].0) ,[NEQ(Mon_Tank_Destination,2) NEQ(Mon_Tank_Destination,3) ,EQU(Mon_Tank_Destination,3) EQU(MON_VALV_ENBL,1) XIO(W4303_Pump.I_Running) ,XIC(Drum_Transfer) ] OTU(Task_Permissive[0].1) ] CLR(Mon_Recirc_Transfer_T430X.Val) ,XIC(Mon_Recirc_Transfer_T430X.Sq.Dn[Mon_Recirc_Transfer_T430X.Val]) ADD(Mon_Recirc_Transfer_T430X.Val,1,Mon_Recirc_Transfer_T430X.Val) ,COP(BLANK64,Mon_Recirc_Transfer_T430X.Sq,1) ,OTL(Mon_Recirc_Transfer_T430X.Sq.Step[Mon_Recirc_Transfer_T430X.Val]) ];
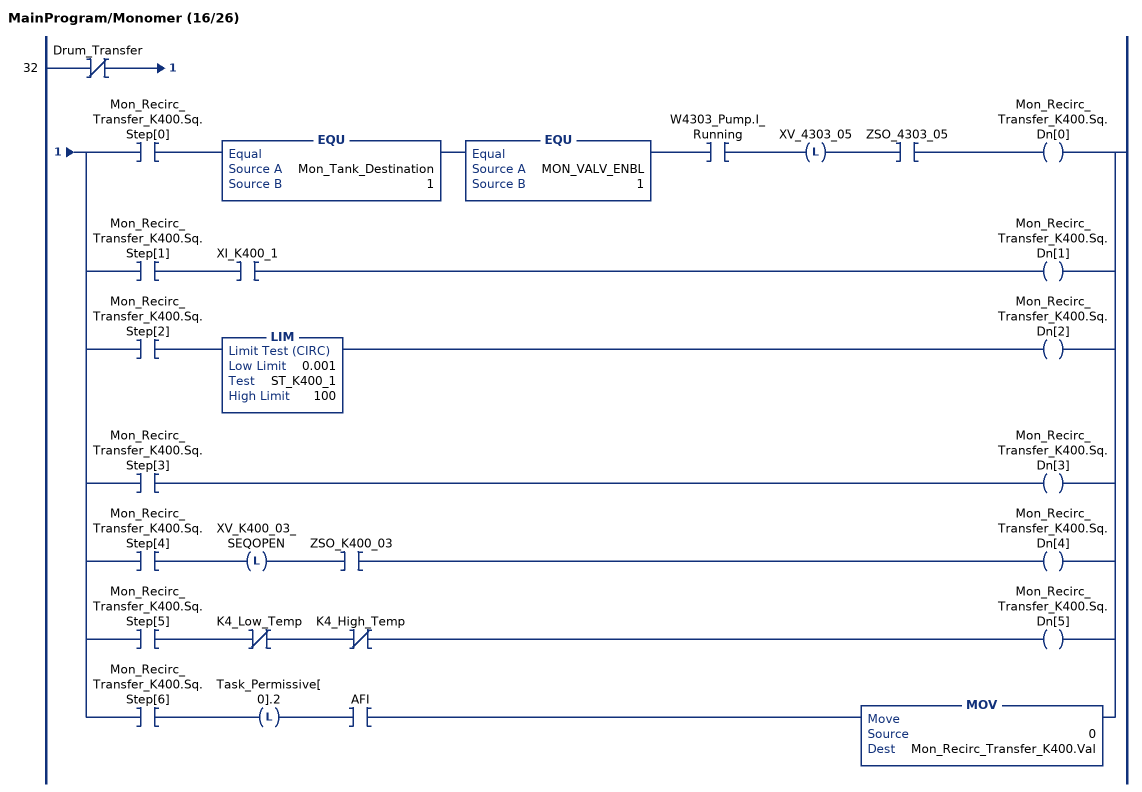
   32: XIO(Drum_Transfer)[XIC(Mon_Recirc_Transfer_K400.Sq.Step[0]) EQU(Mon_Tank_Destination,1) EQU(MON_VALV_ENBL,1) XIC(W4303_Pump.I_Running) OTL(XV_4303_05) XIC(ZSO_4303_05) OTE(Mon_Recirc_Transfer_K400.Sq.Dn[0]) ,XIC(Mon_Recirc_Transfer_K400.Sq.Step[1]) XIC(XI_K400_1) OTE(Mon_Recirc_Transfer_K400.Sq.Dn[1]) ,XIC(Mon_Recirc_Transfer_K400.Sq.Step[2]) LIM(0.001,ST_K400_1,100) OTE(Mon_Recirc_Transfer_K400.Sq.Dn[2]) ,XIC(Mon_Recirc_Transfer_K400.Sq.Step[3]) OTE(Mon_Recirc_Transfer_K400.Sq.Dn[3]) ,XIC(Mon_Recirc_Transfer_K400.Sq.Step[4]) OTL(XV_K400_03_SEQOPEN) XIC(ZSO_K400_03) OTE(Mon_Recirc_Transfer_K400.Sq.Dn[4]) ,XIC(Mon_Recirc_Transfer_K400.Sq.Step[5]) XIO(K4_Low_Temp) XIO(K4_High_Temp) OTE(Mon_Recirc_Transfer_K400.Sq.Dn[5]) ,XIC(Mon_Recirc_Transfer_K400.Sq.Step[6]) OTL(Task_Permissive[0].2) XIC(AFI) MOV(0,Mon_Recirc_Transfer_K400.Val) ];
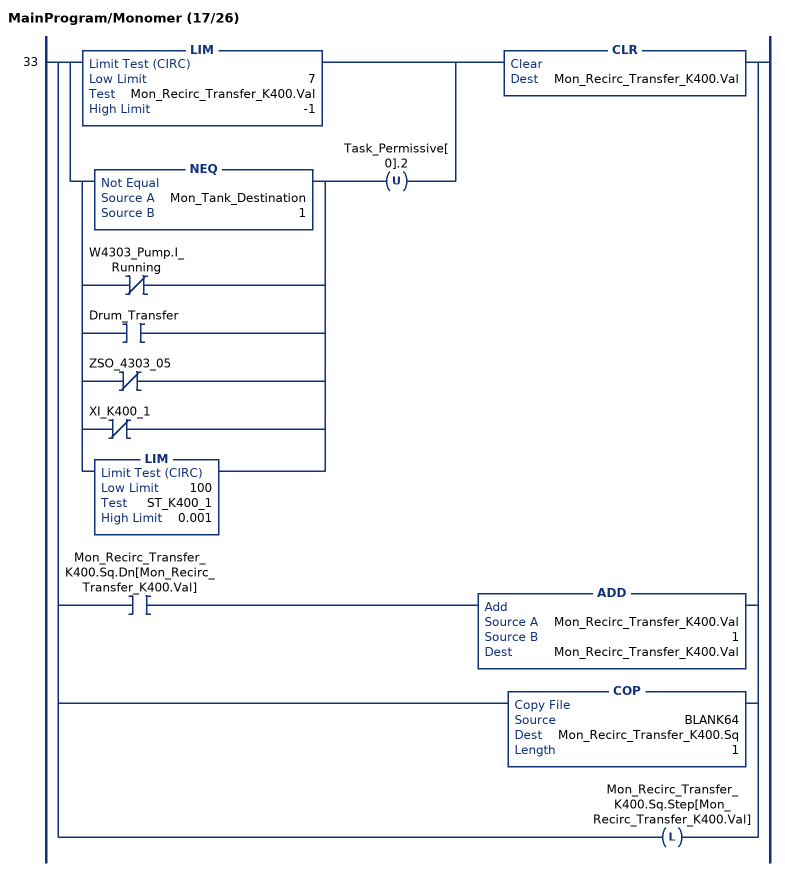
   33: [[LIM(7,Mon_Recirc_Transfer_K400.Val,-1) ,[NEQ(Mon_Tank_Destination,1) ,XIO(W4303_Pump.I_Running) ,XIC(Drum_Transfer) ,XIO(ZSO_4303_05) ,XIO(XI_K400_1) ,LIM(100,ST_K400_1,0.001) ] OTU(Task_Permissive[0].2) ] CLR(Mon_Recirc_Transfer_K400.Val) ,XIC(Mon_Recirc_Transfer_K400.Sq.Dn[Mon_Recirc_Transfer_K400.Val]) ADD(Mon_Recirc_Transfer_K400.Val,1,Mon_Recirc_Transfer_K400.Val) ,COP(BLANK64,Mon_Recirc_Transfer_K400.Sq,1) ,OTL(Mon_Recirc_Transfer_K400.Sq.Step[Mon_Recirc_Transfer_K400.Val]) ];
